SUBAPPLICATION Uebung_011a2_AX (* Numeric Value Output und BUTTON_PRESS_REPEAT_DONE *)
  (* Standard: 61499-2; Description: Copyright (c) 2023 Meisterschulen am Ostbahnhof This program and the accompanying materials are made available under the terms of the Eclipse Public License 2.0 which is available at https://www.eclipse.org/legal/epl-2.0/ SPDX-License-Identifier: EPL-2.0 *)
  (* Version 1.0, 2023-10-23, Franz Höpfinger, Meisterschulen am Ostbahnhof, initial API and implementation and/or initial documentation *)
  PACKAGE Uebungen;
  IMPORT Uebungen::const::UT::DefaultPool::OutputNumber_N1;
  IMPORT logiBUS::io::DI::logiBUS_DI::Input_I1;
  IMPORT logiBUS::io::DI::logiBUS_DI_Events::BUTTON_LONG_PRESS_UP;
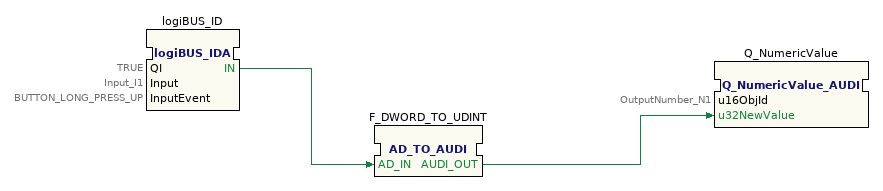
  (* BUTTON_PRESS_UP BUTTON_LONG_PRESS_HOLD BUTTON_LONG_PRESS_UP *)
  FBS
    Q_NumericValue : isobus::UT::Q::Q_NumericValue_AUDI(u16ObjId := OutputNumber_N1);
    logiBUS_ID : logiBUS::io::DI::logiBUS_IDA(QI := TRUE, Input := Input_I1, InputEvent := BUTTON_LONG_PRESS_UP);
    F_DWORD_TO_UDINT : adapter::conversion::unidirectional::AD_TO_AUDI;
  END_FBS
  ADAPTER_CONNECTIONS
    logiBUS_ID.IN TO F_DWORD_TO_UDINT.AD_IN;
    F_DWORD_TO_UDINT.AUDI_OUT TO Q_NumericValue.u32NewValue;
  END_CONNECTIONS
END_SUBAPPLICATION
